FUNCTION_BLOCK FB_WashingPhase

VAR_INPUT
END_VAR

VAR_OUTPUT
	bWashingDone 	: BOOL; 	//washing done flag
	bWashingError 	: BOOL;		//washing error flag
END_VAR

VAR
END_VAR

//bWashingDone := //Verdadeiro quando a etapa de lavagem for concluída

END_FUNCTION_BLOCK

(* stored: Version 1.1.0.1, ProductVersion 3.1.4024.12
   POU FB_WashingPhase: Id {8cd1e697-bf8b-43c9-9f41-396622ef9579}, SpecialFunc None *)
